FUNCTION_BLOCK Performance10 (* Composite Function Block Type *)
  (* Standard: 61499-2 *)
  (* Version 1.0, 2020-12-26, jetbrains *)
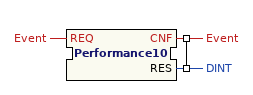
  EVENT_INPUT
    REQ; (* Normal Execution Request *)
  END_EVENT
  EVENT_OUTPUT
    CNF WITH RES; (* Execution Confirmation *)
  END_EVENT
  VAR_OUTPUT
    RES : DINT; (* Output event qualifier *)
  END_VAR
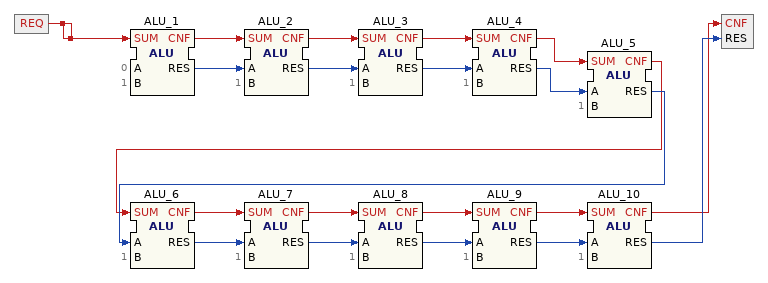
  FBS
    ALU_1 : ALU(A := 0, B := 1);
    ALU_2 : ALU(B := 1);
    ALU_3 : ALU(B := 1);
    ALU_4 : ALU(B := 1);
    ALU_5 : ALU(B := 1);
    ALU_9 : ALU(B := 1);
    ALU_8 : ALU(B := 1);
    ALU_10 : ALU(B := 1);
    ALU_7 : ALU(B := 1);
    ALU_6 : ALU(B := 1);
  END_FBS
  EVENT_CONNECTIONS
    REQ TO ALU_1.SUM;
    ALU_1.CNF TO ALU_2.SUM;
    ALU_2.CNF TO ALU_3.SUM;
    ALU_3.CNF TO ALU_4.SUM;
    ALU_4.CNF TO ALU_5.SUM;
    ALU_6.CNF TO ALU_7.SUM;
    ALU_10.CNF TO CNF;
    ALU_7.CNF TO ALU_8.SUM;
    ALU_8.CNF TO ALU_9.SUM;
    ALU_9.CNF TO ALU_10.SUM;
    REQ TO ALU_1.SUM;
    ALU_5.CNF TO ALU_6.SUM;
  END_CONNECTIONS
  DATA_CONNECTIONS
    ALU_1.RES TO ALU_2.A;
    ALU_2.RES TO ALU_3.A;
    ALU_3.RES TO ALU_4.A;
    ALU_4.RES TO ALU_5.A;
    ALU_8.RES TO ALU_9.A;
    ALU_6.RES TO ALU_7.A;
    ALU_7.RES TO ALU_8.A;
    ALU_9.RES TO ALU_10.A;
    ALU_5.RES TO ALU_6.A;
    ALU_10.RES TO RES;
  END_CONNECTIONS
END_FUNCTION_BLOCK
